{attribute addProperty BoxType "EL2642-0000-0016"}
{attribute addProperty Id "Device_statusAT %I*Device_status_A35574DA162"}
{attribute addProperty CRC "2070112929"}
{attribute addProperty SizeInBites "16"}
{attribute addProperty SizeInBytes "2"}
TYPE DO_Inputs_Device_7B636AA1 :
STRUCT
	{attribute addProperty Name "Device_status"}
	Device_status AT %I* : Device_status_A35574DA;
END_STRUCT
END_TYPE

(* stored: Version 1.2.0.0, ProductVersion 3.1.4024.9
   DUT DO_Inputs_Device_7B636AA1: Id {2736b577-3568-4fb2-9f82-32fd2805454b} *)
